TYPE TcoUrEseries_IO_v_1_x_x :
STRUCT
	PnIoBoxState AT %I*	:	UINT;
	PnIoBoxDiag AT %I*	:	UINT;
	PnIoBoxCtrl AT %Q*	:	UINT;
	{attribute addProperty Name "<#IN#>"}
	In : TcoUrCb3_Inputs_v_3_x_x;
	{attribute addProperty Name "<#OUT#>"}
	Out : TcoUrCb3_Outputs_v_3_x_x;
END_STRUCT
END_TYPE

(* stored: Version 1.1.0.1, ProductVersion 3.1.4024.12
   DUT TcoUrEseries_IO_v_1_x_x: Id {4c851940-ef1d-0a11-32ea-0de9b12b8434} *)
